FUNCTION THRHOLD : BOOL
VAR_INPUT
	
	A : REAL;
	B : REAL;
	THRESH: REAL:= 0.1;
END_VAR
VAR
END_VAR


 THRHOLD :=(ABS(A -B) < THRESH);

END_FUNCTION

(* stored: Version 1.1.0.1
   POU THRHOLD: Id {acfced55-1709-482e-bc9e-3cb78e1b4e95}, SpecialFunc None *)
